// TIA Portal V18 export
FUNCTION "_screenTargetUtility" : Void   // FC28, FBD
{ S7_Optimized_Access := 'TRUE' }
VERSION : 0.1
// stored: AutoNumber true, IsIECCheckEnabled false, SetENOAutomatically false, UDAEnableTagReadback false
   VAR_INPUT
      "M" : "axis_FBD";
   END_VAR
   VAR_OUTPUT
      t_ax : "hmi_home_1";
      h_ax : "hmi_home_1";
   END_VAR
BEGIN

REGION Network 1 (SCL)
   #h_ax.eF := #M.s_fwd_ind;
   #h_ax.eR := #M.s_rev_ind;
   #h_ax.mF := #M.s_fwd_mechOK;
   #h_ax.mR := #M.s_rev_mecOK;
   #h_ax.pos := #M.POS;

   #t_ax.pos := #M.AMANGRDB.aut_target;
END_REGION
END_FUNCTION
